Staubli VAL3: FrameItem.dtx

public frame fFrame = {fatherId=world[0]}
public pointRx pO = {fatherId=world[0]}
public pointRx pX = {fatherId=world[0]}
public pointRx pY = {fatherId=world[0]}
public string sName
